Universal Robots PolyScope program: FlexibleEthernetIpExample.urp

Program FlexibleEthernetIpExample (installation=default directory=/programs/usbdisk createdIn=5.19.0 lastSavedIn=5.19.0 robotSerialNumber=20195399999)
Calibrated DH parameters: a=[0, -0.24355, -0.2132, 0, 0, 0]; d=[0.15185, 0, 0, 0.13105, 0.08535, 0.0921]; alpha=[1.570796, 0, 0, 1.570796, -1.570796, 0]; deltaTheta=[0, 0, 0, 0, 0, 0]
InitVariablesNode
BeforeStart
  Script file /programs/usbdisk/FlexibleEthernetIp.script
    | ###################################################################################################################################
    | # Performance It is recommended to consider performance limitation before integrating custom Ethernet/IP Adapter with PLC Scanner.
    | # All read and write operations are delegated to non-realtime threads.
    | # In internal tests write/read turnaround cycle with PLC RPI set to 5ms wasonaverage40ms,maximumat90ms.
    | # At this point it is not recommended to use custom assemblies for applications requiring RPI below 20ms.
    | ###################################################################################################################################
    | #
    | # Generated script with URManager https://github.com/2onk/UR_Manager
    | # Feel free to contact me Sadek, David dasa@universal-robots.com
    | # V1.0 - 11.11.2024
    | ###########################################################################
    | 
    | ###
    | # Function creates new configuration in EIP Adapter
    | # NOTE: Configurations can not be changed
    | # Ethernet/IP adapter needs to be restarted to clear all configurations
    | # Configuration needs to be added before connection from Ethernet/IP scanner is activated.
    | #
    | # Stops program if configuration adding fails
    | # @param robot_to_scanner int instance id for T->O
    | # @param scanner_to_robot int instance id for O->T
    | # @param size int size of each of the instances
    | ###
    | def eip_register_connection(robot_to_scanner = 101, robot_to_scanner_size = 1, scanner_to_robot = 111, scanner_to_robot_size = 1):
    |   local eip_configurator = rpc_factory("xmlrpc", "http://127.0.0.1:40000/RPC2")
    |   if(not eip_configurator.add_configuration(robot_to_scanner, robot_to_scanner_size, scanner_to_robot, scanner_to_robot_size)):
    |     popup("Adding Flexible Ethernet IP instances failed")
    |     halt
    |   end
    |   eip_configurator.closeXMLRPCClientConnection()
    |   sleep(1.0)
    | end
    | 
    | # Variable is set to True after custom Ethernet/IP instances are configurad
    | # It can be used in threads started before configuraiton function is called
    | global eip_configured = False
    | 
    | ###
    | # Create mapping between Ethernet/IP registers and named variables
    | # note: function has to be called after configuration and before any other function
    | #
    | # @param robot_to_scanner string instance id for T->O
    | # @param scanner_to_robot string instance id for O->T
    | # @param size int size of each of the instances
    | ###
    | def init_eip_communication(robot_to_scanner = "101", scanner_to_robot = "111", robot_to_scanner_size = 1, scanner_to_robot_size = 1):
    |   global robotOutputs = eip_writer_factory(robot_to_scanner, robot_to_scanner_size)
    |   global robotInputs = eip_reader_factory(scanner_to_robot, scanner_to_robot_size)
    | 
    |   ##########################
    |   # in Scanner T2O, robot to Scanner
    |   ##########################
    | 
    |   robotInputs.define_bit(0, 0, "Byte0_Bit0")
    |   robotInputs.define_bit(0, 1, "Byte0_Bit1")
    |   robotInputs.define_bit(0, 2, "Byte0_Bit2")
    |   robotInputs.define_bit(0, 3, "Byte0_Bit3")
    |   robotInputs.define_bit(0, 4, "Byte0_Bit4")
    |   robotInputs.define_bit(0, 5, "Byte0_Bit5")
    |   robotInputs.define_bit(0, 6, "Byte0_Bit6")
    |   robotInputs.define_bit(0, 7, "Byte0_Bit7")
    | 
    | 
    |   ##########################
    |   # in Scanner O2T, Scanner to robot
    |   ##########################
    |   robotOutputs.define_bit(0, 0, "Byte0_Bit0")
    |   robotOutputs.define_bit(0, 1, "Byte0_Bit1")
    |   robotOutputs.define_bit(0, 2, "Byte0_Bit2")
    |   robotOutputs.define_bit(0, 3, "Byte0_Bit3")
    |   robotOutputs.define_bit(0, 4, "Byte0_Bit4")
    |   robotOutputs.define_bit(0, 5, "Byte0_Bit5")
    |   robotOutputs.define_bit(0, 6, "Byte0_Bit6")
    |   robotOutputs.define_bit(0, 7, "Byte0_Bit7")
    | 
    | 
    |   # Watchdog will pause program after 1s of no communication from Scanner
    |   robotInputs.set_watchdog(1, 1)
    | 
    |   # Set all output bits to 0
    |   robotOutputs.clear()
    | 
    |   global eip_configured = True
    | end
    | 
    | ##########################################################################################
    | # In the following lines you will find example methods to customize your Input variables
    | ##########################################################################################
    | 
    | ###
    | # Add custom field of type REAL.
    | #
    | # @param name string name
    | # @param offset int offset Starting offset in Scanner
    | ###
    | def add_custom_real(name, offset):
    |   robotInputs.define_float32(offset, name)
    | end
    | 
    | ###
    | # Add custom field of type WORD.
    | # Additional field should be configured on Scanner.
    | #
    | # @param name string name
    | # @param offset int offset Starting offset in Scanner
    | ###
    | def add_custom_word(name, offset):
    |   robotInputs.define_uint16(offset, name)
    | end
    | 
    | ###
    | # Add custom field of type BYTE.
    | # Additional field should be configured on Scanner.
    | #
    | # @param name string name
    | # @param offset int offset Starting offset in Scanner
    | ###
    | def add_custom_byte(name, offset):
    |   robotInputs.define_uint8(offset, name)
    | end
    | 
    | ###
    | # Example for reading custom offset from user parameter on Scanner
    | # Custom offset can be written to user register by ansi program
    | # Custom variable name is defined with add_custom_real function
    | # @returns number custom variable value. Type depends on the defined value type.
    | ###
    | def get_custom_variable(name):
    |   return robotInputs.read(name)
    | end
    | 
    | 
    | ###
    | # Read example inputs
    | #
    | ###
    | def read_example_inputs():
    |     local example_struct = robotInputs.read(["Byte0_Bit0", "Byte0_Bit1"])
    |     if(example_struct.Byte0_Bit0):
    |         textmsg("Byte0_Bit0 is True")
    |     elif(example_struct.Byte0_Bit1):
    |         textmsg("Byte0_Bit1 is True")
    |     end
    | end
    | 
    | ##########################################################################################
    | # In the following lines you will find example methods to customize your Output variables
    | ##########################################################################################
    | 
    | ###
    | # Set and reset example bits
    | #
    | ###
    | def set_example_eip_outputs():
    |   robotOutputs.write(struct(Byte0_Bit0 = True))
    |   sleep(2)
    |   robotOutputs.write(struct(Byte0_Bit0 = False))
    |   sleep(2)
    |   robotOutputs.write(struct(Byte0_Bit1 = True))
    |   sleep(2)
    |   robotOutputs.write(struct(Byte0_Bit1 = False))
    | end
  Script: eip_register_connection()
  Script: init_eip_communication()
  'Set your example InputByte0 starting with byte offset 0'
  Script: add_custom_byte("InputByte0",0)
Robot Program (runOnlyOnce=false)
  Folder Set_Output_example
    'Set some example outputs to scanner'
    Script: set_example_eip_outputs()
  Folder Read_custom_byte
    'read your customized InputByte0 as byte in decimal'
    eip_in_byte := get_custom_variable("InputByte0")
  Folder Read_input_bits
    'read example scanner outputs and print the in log history'
    Script: read_example_inputs()
